(* PLC project Unnamed, Unknown Unnamed 1 *)
(* stored: creationDateTime 2026-02-02T20:10:37, modificationDateTime 2026-02-02T20:33:21 *)

PROGRAM program0
  VAR
    Fault AT %IX0.3 : BOOL;
    Reset AT %IX0.1 : BOOL;
    MaintenanceAlert AT %QX0.2 : BOOL;
    Counter AT %QX0.3 : INT;
  END_VAR
  VAR
    CTU0 : CTU;
  END_VAR
  VAR  (* added by the conversion: wires and edge detectors of the diagram *)
    R_TRIG1 : R_TRIG;
    R_TRIG2 : R_TRIG;
  END_VAR

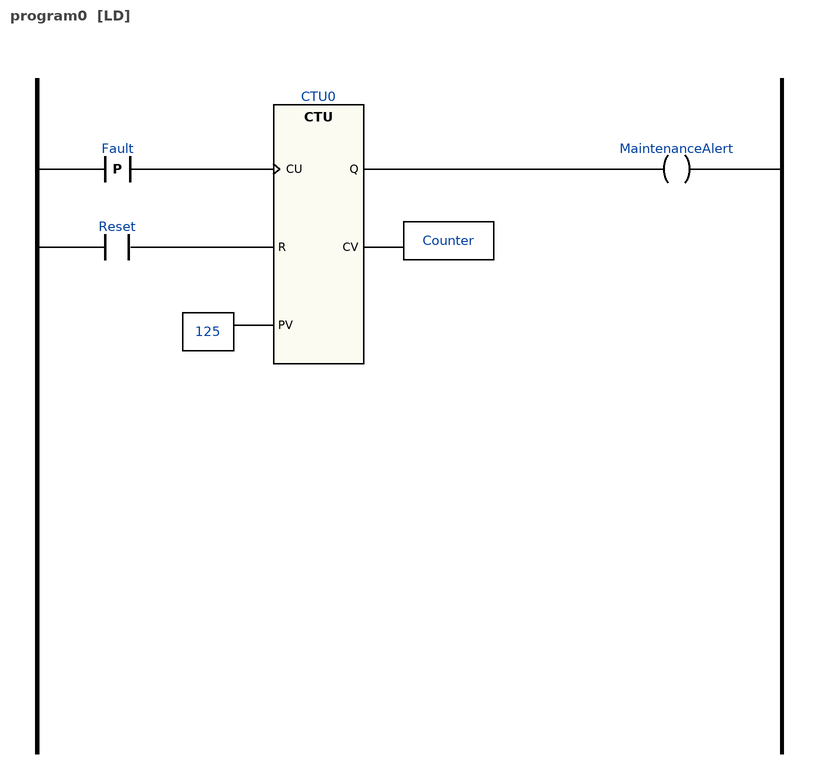
(* LD diagram, written out as Structured Text *)
R_TRIG1(CLK := Fault);
R_TRIG2(CLK := R_TRIG1.Q);
CTU0(CU := R_TRIG2.Q, R := Reset, PV := 125);
MaintenanceAlert := CTU0.Q;
Counter := CTU0.CV;
END_PROGRAM

CONFIGURATION Config0
  RESOURCE Res0 ON PLC
    TASK task0(INTERVAL := T#20ms, PRIORITY := 0);
    PROGRAM instance0 WITH task0 : program0;
  END_RESOURCE
END_CONFIGURATION
